PROGRAM PRG_DoSomeMath
VAR_INPUT
	
END_VAR
VAR
	rVariable1 : REAL;
	rVariable2 : REAL;
	rVariable3 : REAL;
	rVariable4 : REAL;
	rPRG_Count : UINT;
END_VAR

rPRG_Count := rPRG_Count + 1;

rVariable1 := F_AdditionFunction(23.23,4.3);
rVariable2 := F_SubstractFunction(23.23,4.3);
rVariable3 := F_MultiplicationFunction(23.23,4.3);
rVariable4 := F_DivisionFunction(23.23,4.3);

END_PROGRAM

(* stored: Version 1.1.0.1, ProductVersion 3.1.4024.13
   POU PRG_DoSomeMath: Id {c41a72ce-b66f-42f8-8b8f-d85cb77cd985}, SpecialFunc None *)
